FUNCTION_BLOCK fbStackerServo implements ITFServoMotor
VAR_INPUT
END_VAR
VAR_OUTPUT
END_VAR
VAR
	
	IPositie : INT;
	TONBeweegTimer : TON;
	BTONVariabele : BOOL;
	EMotorStatusIntern : E_MotorStatus;
	IDoelPositie	: INT;
	BInternEnable : BOOL;
	
	MotorStatusString: STRING;
END_VAR

MotorStatusString := TO_STRING(EMotorStatusIntern);

METHOD PUBLIC BeweegNaarDoel
VAR_INPUT

END_VAR

VAR CONSTANT
	IMotorSnelheid : INT := 1; 
	IMotorStopSnelheid : INT:= 5;
END_VAR

//notes
//  status schrijven en
VAR
	BBewegenActief: BOOL;
END_VAR
(* ================= TIMER ================= *)
TONBeweegTimer(
    IN := BInternEnable AND NOT BBewegenActief,
    PT := T#0.3S
);

(* ================= START NA TIMER ================= *)
IF TONBeweegTimer.Q THEN
    BBewegenActief := TRUE;
    TONBeweegTimer(IN := FALSE);   // DIRECT reset → cruciaal
END_IF

(* ================= STATUS ================= *)
IF BInternEnable THEN
    EMotorStatusIntern := 1;
ELSE
    EMotorStatusIntern := 0;
END_IF

(* ================= BEWEGEN ================= *)
IF BInternEnable AND BBewegenActief THEN

    IF IDoelPositie > IPositie THEN
        IPositie := IPositie + IMotorSnelheid;
        EMotorStatusIntern := 3;

        IF IPositie >= IDoelPositie THEN
            IPositie := IDoelPositie;
            BBewegenActief := FALSE;
        END_IF

    ELSIF IDoelPositie < IPositie THEN
        IPositie := IPositie - IMotorSnelheid;
        EMotorStatusIntern := 4;

        IF IPositie <= IDoelPositie THEN
            IPositie := IDoelPositie;
            BBewegenActief := FALSE;
        END_IF

    ELSE
        BBewegenActief := FALSE;
    END_IF
END_IF

(* ================= UIT / STOP ================= *)
IF NOT BInternEnable THEN
    BBewegenActief := FALSE;
    TONBeweegTimer(IN := FALSE);

    IF IPositie > 0 THEN
        IPositie := IPositie - IMotorStopSnelheid;
        IF IPositie < 0 THEN IPositie := 0; END_IF

    ELSIF IPositie < 0 THEN
        IPositie := IPositie + IMotorStopSnelheid;
        IF IPositie > 0 THEN IPositie := 0; END_IF
    END_IF
END_IF
END_METHOD

PROPERTY DoelPositie : int
GET
doelpositie := idoelpositie;
END_GET
SET
idoelpositie := doelpositie;
END_SET
END_PROPERTY

PROPERTY Enable : bool
GET
Enable := BInternEnable;
END_GET
SET
BInternEnable:= Enable;
END_SET
END_PROPERTY

PROPERTY MotorStatus : E_MotorStatus
GET
MotorStatus:=  EMotorStatusIntern;
END_GET
SET
EMotorStatusIntern := MotorStatus;
END_SET
END_PROPERTY

PROPERTY Positie : INT
GET
positie:= IPositie;
END_GET
END_PROPERTY

END_FUNCTION_BLOCK

(* stored: Version 1.1.0.1
   POU fbStackerServo: Id {63955412-bcd3-4783-ab58-d217a713d49f}, SpecialFunc None
   Method BeweegNaarDoel: Id {3aa19c92-d64d-4fa9-b144-f711e11a9595}
   Property DoelPositie: Id {bcaa4272-0182-490b-b5c5-17ac81e472ef}
   Get Get: Id {e42b4d98-7528-4ccf-bc6d-8dd18947a815}
   Set Set: Id {96a1827d-06a7-4211-a2e1-0f154c576779}
   Property Enable: Id {ce81a4dc-e68d-4ced-817d-12d70bcc0997}
   Get Get: Id {23006fc9-e0d1-4516-a217-ab21628f28b3}
   Set Set: Id {127d2ac9-0d45-4fcb-bb22-ff7dc6826e0e}
   Property MotorStatus: Id {f3515037-d7f1-4cdf-986c-5e4909665074}
   Get Get: Id {27bff63a-6d8b-446e-b4a2-550c7791f64a}
   Set Set: Id {b4817821-45b4-4de7-bd99-86450dd53a84}
   Property Positie: Id {3f190714-8df9-4d2a-abfe-e5a5df771a72}
   Get Get: Id {2efa94e1-195f-4ab4-81b1-0730edbf470f} *)
